DATA_BLOCK "DB_MESLoadData"
{ S7_Optimized_Access := 'TRUE' }
VERSION : 0.1
// ATTRIBUTES
// AUTO_NUMBER = False
// BLOCK_NUMBER = 2800
// END_ATTRIBUTES
   VAR
      Station1 : "UDT_MESLoadData";
      Station2 : "UDT_MESLoadData";
      Station3 : "UDT_MESLoadData";
      Station4 : "UDT_MESLoadData";
   END_VAR


BEGIN

END_DATA_BLOCK

